KUKA KRL data list: kurostream.dat

&ACCESS RVP
&REL 219
&PARAM TEMPLATE = C:\KRC\Roboter\Template\vorgabe
&PARAM EDITMASK = *
DEFDAT KUROSTREAM

DECL char mh_sensorname[10] = "Kurostream"

INT mh_response_stream_ms = 12
INT mh_waitfordata_ms = 12
INT mh_robot_status	= 0
INT	mh_in_traject_id = 0
INT	mh_out_traject_id = 0
INT mh_frame_type = 1
ENDDAT
